# B&R Automation Studio project Panasonic_LinkaPowerCP2_A2021055 (part 42)

#### Main.st - Init, cyclic, exit code
```iecst
PROGRAM _INIT
	(* Insert code here *)
	SKTcpClientTrace_1.Params.IPportClient := 15000;
	SKTcpClientTrace_1.Cmd.LoggerOn:= FALSE;
END_PROGRAM

PROGRAM _CYCLIC

	//Priradenie indexu paletky//
    a:= P2_StoperZaklTesnenia.PAR.CisloPaletky;
	P2_StoperZaklTesnenia.PAR.CisloPaletky_STRING:= USINT_TO_STRING(a);

    //Parametre komunikácie//
    memcpy(ADR(SKTcpClientTrace_1.Params.IPaddrServ),ADR('192.168.128.250'),SIZEOF('192.168.128.250'));

    SKTcpClientTrace_1.Params.IPportServ := 12000;

	SKTcpClientTrace_1.pDevice := ADR('HDD_LOGGER');
	SKTcpClientTrace_1.pFile := ADR('logger_sktcpclienttrace_3.log');
    SKTcpClientTrace_1();

    //Parametre komunikácie//
    //Vstupy pre server//
    SKTcpClientTrace_1.Params.Packet.type := TRCB_P2_ZakladacTesnenia_ST3.INPUTS.TYP_Prikazu;
    SKTcpClientTrace_1.Params.Packet.workplace := TRCB_P2_ZakladacTesnenia_ST3.INPUTS.CisloStanice;
    SKTcpClientTrace_1.Params.Packet.rfid := TRCB_P2_ZakladacTesnenia_ST3.INPUTS.CisloPaletky;
    SKTcpClientTrace_1.Params.Packet.master := TRCB_P2_ZakladacTesnenia_ST3.INPUTS.QRkodPowerCP;
    SKTcpClientTrace_1.Params.Packet.dps1:= TRCB_P2_ZakladacTesnenia_ST3.INPUTS.QRkodFiltra;
    SKTcpClientTrace_1.Params.Packet.dps2:= '';
    SKTcpClientTrace_1.Params.Packet.dps3:= '';
    SKTcpClientTrace_1.Params.Packet.dps4:= '';
    SKTcpClientTrace_1.Params.Packet.dps5:= '';
    SKTcpClientTrace_1.Params.Packet.operator_id := TRCB_P2_ZakladacTesnenia_ST3.INPUTS.ID_Operatora;
    SKTcpClientTrace_1.Params.Packet.data_report:= TRCB_P2_ZakladacTesnenia_ST3.INPUTS.Report;
    SKTcpClientTrace_1.Params.Packet.result := TRCB_P2_ZakladacTesnenia_ST3.INPUTS.StavPaletky;

    //Výstupy zo servera//
    TRCB_P2_ZakladacTesnenia_ST3.OUTPUTS.TYP_Prikazu:= SKTcpClientTrace_1.Internal.Splitter.out[1];
    TRCB_P2_ZakladacTesnenia_ST3.OUTPUTS.CisloStanice:= SKTcpClientTrace_1.Internal.Splitter.out[2];
    TRCB_P2_ZakladacTesnenia_ST3.OUTPUTS.CisloPaletky:= SKTcpClientTrace_1.Internal.Splitter.out[3];
    IF TRCB_P2_ZakladacTesnenia_ST3.INPUTS.TYP_Prikazu = '0' THEN
        TRCB_P2_ZakladacTesnenia_ST3.OUTPUTS.CisloEtikety:= SKTcpClientTrace_1.Internal.Splitter.out[4];
    ELSE
        TRCB_P2_ZakladacTesnenia_ST3.OUTPUTS.QRkodPowerCP:= SKTcpClientTrace_1.Internal.Splitter.out[4];
    END_IF
    TRCB_P2_ZakladacTesnenia_ST3.OUTPUTS.QRkodFiltra:= SKTcpClientTrace_1.Internal.Splitter.out[5];
    TRCB_P2_ZakladacTesnenia_ST3.OUTPUTS.ID_Operatora:= SKTcpClientTrace_1.Internal.Splitter.out[10];
    TRCB_P2_ZakladacTesnenia_ST3.OUTPUTS.DruhCinnostiNaPaletke:= SKTcpClientTrace_1.Internal.Splitter.out[11];
    TRCB_P2_ZakladacTesnenia_ST3.OUTPUTS.PovolenieCinnostiNaPaletke:= SKTcpClientTrace_1.Internal.Splitter.out[12];

    //Volanie funkcie SequenceControl//
    SequenceControl(SC:= SC_KOM_Server);

    CASE SC_KOM_Server.Step OF

        0:
            SC_KOM_Server.StepName:= '0 - Nulovanie';
            SKTcpClientTrace_1.Cmd.Send:= FALSE;
            TRCB_P2_ZakladacTesnenia_ST3.CMD.VyziadajStavPaletky_TYP1:= FALSE;
            TRCB_P2_ZakladacTesnenia_ST3.CMD.PriradQRkodFiltra_TYP3:= FALSE;
            TRCB_P2_ZakladacTesnenia_ST3.CMD.VyziadajCisloEtikety_TYP0:= FALSE;
			TRCB_P2_ZakladacTesnenia_ST3.CMD.OdosliStavPaletky_TYP2:= FALSE;
			TRCB_P2_ZakladacTesnenia_ST3.CMD.VyziadajStavPanatrace_TYP4:= FALSE;
            TRCB_P2_ZakladacTesnenia_ST3.STATUS.KomunikaciaUkoncena:= FALSE;
			TRCB_P2_ZakladacTesnenia_ST3.STATUS.KomunikaciaError:= FALSE;
			TRCB_P2_ZakladacTesnenia_ST3.STATUS.KOM_READY:= FALSE;
            PocetDopytovNaServer:= 0;

            IF SKTcpClientTrace_1.Internal.Step = 0 THEN
                SKTcpClientTrace_1.Enable:= TRUE;
                SC_KOM_Server.ResetStep:= TRUE;
                SC_KOM_Server.Step:= 1;
            ELSIF SKTcpClientTrace_1.Internal.Step = 15 THEN
                SKTcpClientTrace_1.Enable:= TRUE;
                SC_KOM_Server.ResetStep:= TRUE;
                SC_KOM_Server.Step:= 1;
            ELSE
                SKTcpClientTrace_1.Enable:= FALSE;
            END_IF

        1:
            SC_KOM_Server.StepName:= '1 - Rozhodnutie o cinnosti';
            TRCB_P2_ZakladacTesnenia_ST3.STATUS.KOM_READY:= TRUE;
			IF TRCB_P2_ZakladacTesnenia_ST3.CMD.VyziadajStavPaletky_TYP1 THEN
                TRCB_P2_ZakladacTesnenia_ST3.STATUS.KOM_READY:= FALSE;
				SC_KOM_Server.Step:= 10;
            ELSIF TRCB_P2_ZakladacTesnenia_ST3.CMD.PriradQRkodFiltra_TYP3 THEN
                TRCB_P2_ZakladacTesnenia_ST3.STATUS.KOM_READY:= FALSE;
				SC_KOM_Server.Step:= 20;
            ELSIF TRCB_P2_ZakladacTesnenia_ST3.CMD.VyziadajCisloEtikety_TYP0 THEN
                TRCB_P2_ZakladacTesnenia_ST3.STATUS.KOM_READY:= FALSE;
				SC_KOM_Server.Step:= 30;
            ELSIF TRCB_P2_ZakladacTesnenia_ST3.CMD.OdosliStavPaletky_TYP2 THEN
				TRCB_P2_ZakladacTesnenia_ST3.STATUS.KOM_READY:= FALSE;
				SC_KOM_Server.Step:= 40;
			ELSIF TRCB_P2_ZakladacTesnenia_ST3.CMD.VyziadajStavPanatrace_TYP4 THEN
				TRCB_P2_ZakladacTesnenia_ST3.STATUS.KOM_READY:= FALSE;
				SC_KOM_Server.Step:= 50;
            END_IF

        10:
            SC_KOM_Server.StepName:= '10 - Vyziadanie stavu paletky - odoslanie dat na server';
            SC_KOM_Server.IdleTime.PT:= T#3s;
            SC_KOM_Server.AlarmTime.PT:= T#10s;
		    SC_KOM_Server.AlarmTime.IN:= TRUE;

			TRCB_P2_ZakladacTesnenia_ST3.INPUTS.CisloPaletky:= 'Pal';
			brsstrcat(ADR(TRCB_P2_ZakladacTesnenia_ST3.INPUTS.CisloPaletky), ADR(P2_StoperZaklTesnenia.PAR.CisloPaletky_STRING));

            TRCB_P2_ZakladacTesnenia_ST3.INPUTS.TYP_Prikazu:= '1';
            TRCB_P2_ZakladacTesnenia_ST3.INPUTS.CisloStanice:= 'ST3';
            TRCB_P2_ZakladacTesnenia_ST3.INPUTS.QRkodPowerCP:= Paletka[a].PAR.QRkodPowerCP;
            TRCB_P2_ZakladacTesnenia_ST3.INPUTS.QRkodFiltra:= '';
            TRCB_P2_ZakladacTesnenia_ST3.INPUTS.ID_Operatora:= Paletka[a].PAR.ID_Operatora;
            TRCB_P2_ZakladacTesnenia_ST3.INPUTS.Report:= '';
            TRCB_P2_ZakladacTesnenia_ST3.INPUTS.StavPaletky:= 'OK';

			IF SKTcpClientTrace_1.Status.staReadyToSend AND NOT SKTcpClientTrace_1.Cmd.Close THEN
				TRCB_P2_ZakladacTesnenia_ST3.OUTPUTS.TYP_Prikazu:= '';
				SKTcpClientTrace_1.Cmd.Send:= TRUE;
				SC_KOM_Server.ResetStep:= TRUE;
				SC_KOM_Server.Step:= 13;
			END_IF

        13:
			SC_KOM_Server.StepName:= '13 - Vyziadanie stavu paletky - odpoved servera';
            SC_KOM_Server.IdleTime.PT:= T#3s;
            SC_KOM_Server.AlarmTime.PT:= T#7s;
            SC_KOM_Server.AlarmTime.IN:= TRUE;

            IF SKTcpClientTrace_1.Status.staReceived AND
                (TRCB_P2_ZakladacTesnenia_ST3.OUTPUTS.TYP_Prikazu = TRCB_P2_ZakladacTesnenia_ST3.INPUTS.TYP_Prikazu) AND
                (TRCB_P2_ZakladacTesnenia_ST3.OUTPUTS.QRkodPowerCP = TRCB_P2_ZakladacTesnenia_ST3.INPUTS.QRkodPowerCP) THEN
                TRCB_P2_ZakladacTesnenia_ST3.STATUS.KomunikaciaUkoncena:= TRUE;
                SC_KOM_Server.ResetStep:= TRUE;
                SC_KOM_Server.Step:= 15;
            ELSIF SC_KOM_Server.AlarmTime.Q AND NOT SKTcpClientTrace_1.Status.staSending THEN
                PocetDopytovNaServer:= PocetDopytovNaServer + 1;
				SKTcpClientTrace_1.Cmd.Close:= TRUE;
				SKTcpClientTrace_1.Cmd.Send:= FALSE;
				SC_KOM_Server.ResetStep:= TRUE;
                SC_KOM_Server.Step:= 14;
            END_IF

        14:
            SC_KOM_Server.StepName:= '14 - Vyziadanie stavu paletky - cakam na opatovny dopyt na server';
            SC_KOM_Server.IdleTime.PT:= T#1s;
            SC_KOM_Server.AlarmTime.PT:= T#10s;
            SC_KOM_Server.IdleTime.IN:= TRUE;

            IF PocetDopytovNaServer < 3 THEN
                IF SC_KOM_Server.IdleTime.Q THEN
                    SC_KOM_Server.ResetStep:= TRUE;
                    SC_KOM_Server.Step:= 10;
                END_IF
            ELSE
                TRCB_P2_ZakladacTesnenia_ST3.STATUS.KomunikaciaError:= TRUE;
                SC_KOM_Server.ResetStep:= TRUE;
                SC_KOM_Server.Step:= 15;
            END_IF

        15:
            SC_KOM_Server.StepName:= '15 - Vyziadanie stavu paletky - cakam na ukoncenie komunikacie';
            SC_KOM_Server.IdleTime.PT:= T#3s;
            SC_KOM_Server.AlarmTime.PT:= T#10s;

            IF NOT TRCB_P2_ZakladacTesnenia_ST3.CMD.VyziadajStavPaletky_TYP1 THEN
                SC_KOM_Server.ResetStep:= TRUE;
                SC_KOM_Server.Step:= 0;
            END_IF

        20:
            SC_KOM_Server.StepName:= '20 - Priradenie QR kodu - odoslanie dat na server';
            SC_KOM_Server.IdleTime.PT:= T#3s;
            SC_KOM_Server.AlarmTime.PT:= T#20s;
            SC_KOM_Server.AlarmTime.IN:= TRUE;

			TRCB_P2_ZakladacTesnenia_ST3.INPUTS.CisloPaletky:= 'Pal';
			brsstrcat(ADR(TRCB_P2_ZakladacTesnenia_ST3.INPUTS.CisloPaletky), ADR(P2_StoperZaklTesnenia.PAR.CisloPaletky_STRING));

            TRCB_P2_ZakladacTesnenia_ST3.INPUTS.TYP_Prikazu:= '3';
            TRCB_P2_ZakladacTesnenia_ST3.INPUTS.CisloStanice:= 'ST3';
            TRCB_P2_ZakladacTesnenia_ST3.INPUTS.QRkodPowerCP:= Paletka[a].PAR.QRkodPowerCP;
            TRCB_P2_ZakladacTesnenia_ST3.INPUTS.QRkodFiltra:= Paletka[a].PAR.QRkodFiltra_5H;
            TRCB_P2_ZakladacTesnenia_ST3.INPUTS.ID_Operatora:= Paletka[a].PAR.ID_Operatora;
            TRCB_P2_ZakladacTesnenia_ST3.INPUTS.Report:= '';
            TRCB_P2_ZakladacTesnenia_ST3.INPUTS.StavPaletky:= 'OK';

			IF SKTcpClientTrace_1.Status.staReadyToSend AND NOT SKTcpClientTrace_1.Cmd.Close THEN
				TRCB_P2_ZakladacTesnenia_ST3.OUTPUTS.TYP_Prikazu:= '';
				SKTcpClientTrace_1.Cmd.Send:= TRUE;
				SC_KOM_Server.ResetStep:= TRUE;
				SC_KOM_Server.Step:= 23;
			END_IF

        23:
            SC_KOM_Server.StepName:= '23 - Priradenie QR kodu - odpoved servera';
			SC_KOM_Server.IdleTime.PT:= T#3s;
            SC_KOM_Server.AlarmTime.PT:= T#7s;
            SC_KOM_Server.AlarmTime.IN:= TRUE;

            IF SKTcpClientTrace_1.Status.staReceived AND
                (TRCB_P2_ZakladacTesnenia_ST3.OUTPUTS.TYP_Prikazu = TRCB_P2_ZakladacTesnenia_ST3.INPUTS.TYP_Prikazu) AND
                (TRCB_P2_ZakladacTesnenia_ST3.OUTPUTS.QRkodPowerCP = TRCB_P2_ZakladacTesnenia_ST3.INPUTS.QRkodPowerCP) THEN
                TRCB_P2_ZakladacTesnenia_ST3.STATUS.KomunikaciaUkoncena:= TRUE;
                SC_KOM_Server.ResetStep:= TRUE;
                SC_KOM_Server.Step:= 25;
            ELSIF SC_KOM_Server.AlarmTime.Q AND NOT SKTcpClientTrace_1.Status.staSending THEN
                PocetDopytovNaServer:= PocetDopytovNaServer + 1;
				SKTcpClientTrace_1.Cmd.Close:= TRUE;
				SKTcpClientTrace_1.Cmd.Send:= FALSE;
				SC_KOM_Server.ResetStep:= TRUE;
                SC_KOM_Server.Step:= 24;
            END_IF

        24:
            SC_KOM_Server.StepName:= '24 - Priradenie QR kodu - cakam na opatovny dopyt na server';
            SC_KOM_Server.IdleTime.PT:= T#1s;
            SC_KOM_Server.AlarmTime.PT:= T#10s;
            SC_KOM_Server.IdleTime.IN:= TRUE;
            SKTcpClientTrace_1.Cmd.Send:= FALSE;

            IF PocetDopytovNaServer < 3 THEN
                IF SC_KOM_Server.IdleTime.Q THEN
                   	SC_KOM_Server.ResetStep:= TRUE;
                    SC_KOM_Server.Step:= 20;
                END_IF
            ELSE
                TRCB_P2_ZakladacTesnenia_ST3.STATUS.KomunikaciaError:= TRUE;
                SC_KOM_Server.ResetStep:= TRUE;
                SC_KOM_Server.Step:= 25;
            END_IF

        25:
            SC_KOM_Server.StepName:= '25 - Priradenie QR kodu - cakam na ukoncenie komunikacie';
            SC_KOM_Server.IdleTime.PT:= T#3s;
            SC_KOM_Server.AlarmTime.PT:= T#10s;

            IF NOT TRCB_P2_ZakladacTesnenia_ST3.CMD.PriradQRkodFiltra_TYP3 THEN
                SC_KOM_Server.ResetStep:= TRUE;
                SC_KOM_Server.Step:= 0;
            END_IF

        30:
            SC_KOM_Server.StepName:= '30 - Vyziadanie serioveho cisla - odoslanie dat na server';
            SC_KOM_Server.IdleTime.PT:= T#3s;
            SC_KOM_Server.AlarmTime.PT:= T#10s;

            TRCB_P2_ZakladacTesnenia_ST3.INPUTS.TYP_Prikazu:= '0';
            TRCB_P2_ZakladacTesnenia_ST3.INPUTS.CisloStanice:= 'ST3';
            TRCB_P2_ZakladacTesnenia_ST3.INPUTS.CisloPaletky;
            TRCB_P2_ZakladacTesnenia_ST3.INPUTS.QRkodPowerCP:= '';
            TRCB_P2_ZakladacTesnenia_ST3.INPUTS.QRkodFiltra:= '';
            TRCB_P2_ZakladacTesnenia_ST3.INPUTS.ID_Operatora:= 'E2';
            TRCB_P2_ZakladacTesnenia_ST3.INPUTS.Report:= '';
            TRCB_P2_ZakladacTesnenia_ST3.INPUTS.StavPaletky:= 'OK';
            SKTcpClientTrace_1.Cmd.Send:= TRUE;

            IF SKTcpClientTrace_1.Cmd.Send AND NOT SKTcpClientTrace_1.Status.staReceived AND NOT SKTcpClientTrace_1.Status.staError THEN
                SC_KOM_Server.ResetStep:= TRUE;
                SC_KOM_Server.Step:= 33;
            END_IF

        33:
            SC_KOM_Server.StepName:= '33 - Vyziadanie serioveho cisla - odpoved servera';
            SC_KOM_Server.IdleTime.PT:= T#3s;
            SC_KOM_Server.AlarmTime.PT:= T#20s;
            SC_KOM_Server.AlarmTime.IN:= TRUE;

            IF SKTcpClientTrace_1.Status.staReceived AND
                (TRCB_P2_ZakladacTesnenia_ST3.OUTPUTS.TYP_Prikazu = TRCB_P2_ZakladacTesnenia_ST3.INPUTS.TYP_Prikazu) THEN
                TRCB_P2_ZakladacTesnenia_ST3.STATUS.KomunikaciaUkoncena:= TRUE;
                SC_KOM_Server.ResetStep:= TRUE;
                SC_KOM_Server.Step:= 35;
            ELSIF SC_KOM_Server.AlarmTime.Q THEN
                TRCB_P2_ZakladacTesnenia_ST3.STATUS.KomunikaciaError:= TRUE;
                SC_KOM_Server.ResetStep:= TRUE;
                SC_KOM_Server.Step:= 35;
            END_IF

        35:
            SC_KOM_Server.StepName:= '35 - Vyziadanie serioveho cisla - cakam na ukoncenie komunikacie';
            SC_KOM_Server.IdleTime.PT:= T#3s;
            SC_KOM_Server.AlarmTime.PT:= T#10s;

            IF NOT TRCB_P2_ZakladacTesnenia_ST3.CMD.VyziadajCisloEtikety_TYP0 THEN
                SC_KOM_Server.ResetStep:= TRUE;
                SC_KOM_Server.Step:= 0;
            END_IF

        40:
            SC_KOM_Server.StepName:= '40 - Odoslanie stavu paletky - odoslanie dat na server';
            SC_KOM_Server.IdleTime.PT:= T#3s;
            SC_KOM_Server.AlarmTime.PT:= T#20s;
            SC_KOM_Server.AlarmTime.IN:= TRUE;

            //Vytvorenie spravy pre report//

            IF NOT SC_KOM_Server.Switch1 THEN
				brsmemset(ADR(Report),0,SIZEOF(Report));
				brsmemset(ADR(TRCB_P2_ZakladacTesnenia_ST3.INPUTS.Report), 0, SIZEOF(TRCB_P2_ZakladacTesnenia_ST3.INPUTS.Report));

				//Kamera 17 - kontrola paletky//
                Report[0].PoradoveCislo:= '1';
                Report[0].Popis:= 'KAM_17_KontrolaPaletky';
                Report[0].FormatHodnoty:= '2';
                Report[0].Tolerancia_MIN_Hodnota:= '';
                Report[0].Tolerancia_MAX_Hodnota:= '';
                Report[0].Nominal:= 'OK';
                Report[0].Tolerancia_MIN_Jednotky:= '';
                Report[0].Tolerancia_MAX_Jednotky:= '';
                IF Reports.Kamery.P2_CAM17_KontrolaPaletky = 'PASS' THEN
                    Report[0].NameranaHodnota:= 'OK';
                ELSE
                    Report[0].NameranaHodnota:= 'NG';
                END_IF
                Report[0].NameranaHodnota_Jednotky:= '';
                Report[0].VyslednyResult:= Reports.Kamery.P2_CAM17_KontrolaPaletky;
                SKTcpClientNewCsvEntry(Report[0].PoradoveCislo,Report[0].Popis,Report[0].FormatHodnoty,Report[0].Tolerancia_MIN_Hodnota,Report[0].Tolerancia_MAX_Hodnota,Report[0].Nominal,Report[0].Tolerancia_MIN_Jednotky,Report[0].Tolerancia_MAX_Jednotky,Report[0].NameranaHodnota,Report[0].NameranaHodnota_Jednotky,Report[0].VyslednyResult, ADR(TRCB_P2_ZakladacTesnenia_ST3.INPUTS.Report));

                //Kamera 1 - kontrola tesnenia//
                Report[1].PoradoveCislo:= '2';
                Report[1].Popis:= 'KAM_1_KontrolaTesnenia';
                Report[1].FormatHodnoty:= '2';
                Report[1].Tolerancia_MIN_Hodnota:= '';
                Report[1].Tolerancia_MAX_Hodnota:= '';
                Report[1].Nominal:= 'OK';
                Report[1].Tolerancia_MIN_Jednotky:= '';
                Report[1].Tolerancia_MAX_Jednotky:= '';
                IF Reports.Kamery.P2_CAM1_KontrolaTesnenia = 'PASS' THEN
                    Report[1].NameranaHodnota:= 'OK';
                ELSE
                    Report[1].NameranaHodnota:= 'NG';
                END_IF
                Report[1].NameranaHodnota_Jednotky:= '';
                Report[1].VyslednyResult:= Reports.Kamery.P2_CAM1_KontrolaTesnenia;
                SKTcpClientNewCsvEntry(Report[1].PoradoveCislo,Report[1].Popis,Report[1].FormatHodnoty,Report[1].Tolerancia_MIN_Hodnota,Report[1].Tolerancia_MAX_Hodnota,Report[1].Nominal,Report[1].Tolerancia_MIN_Jednotky,Report[1].Tolerancia_MAX_Jednotky,Report[1].NameranaHodnota,Report[1].NameranaHodnota_Jednotky,Report[1].VyslednyResult, ADR(TRCB_P2_ZakladacTesnenia_ST3.INPUTS.Report));
                SC_KOM_Server.Switch1:= TRUE;
            END_IF

			TRCB_P2_ZakladacTesnenia_ST3.INPUTS.CisloPaletky:= 'Pal';
			brsstrcat(ADR(TRCB_P2_ZakladacTesnenia_ST3.INPUTS.CisloPaletky), ADR(P2_StoperZaklTesnenia.PAR.CisloPaletky_STRING));

            TRCB_P2_ZakladacTesnenia_ST3.INPUTS.TYP_Prikazu:= '2';
            TRCB_P2_ZakladacTesnenia_ST3.INPUTS.CisloStanice:= 'ST3';
            TRCB_P2_ZakladacTesnenia_ST3.INPUTS.QRkodPowerCP:= Paletka[a].PAR.QRkodPowerCP;
            TRCB_P2_ZakladacTesnenia_ST3.INPUTS.QRkodFiltra:= '';
            TRCB_P2_ZakladacTesnenia_ST3.INPUTS.ID_Operatora:= Paletka[a].PAR.ID_Operatora;
            TRCB_P2_ZakladacTesnenia_ST3.INPUTS.StavPaletky:= Paletka[a].PAR.StavPowerCP;

			IF SKTcpClientTrace_1.Status.staReadyToSend AND NOT SKTcpClientTrace_1.Cmd.Close THEN
				TRCB_P2_ZakladacTesnenia_ST3.OUTPUTS.TYP_Prikazu:= '';
				SKTcpClientTrace_1.Cmd.Send:= TRUE;
				SC_KOM_Server.ResetStep:= TRUE;
				SC_KOM_Server.Step:= 43;
			END_IF

        43:
            SC_KOM_Server.StepName:= '43 - Odoslanie stavu paletky - odpoved servera';
			SC_KOM_Server.IdleTime.PT:= T#3s;
            SC_KOM_Server.AlarmTime.PT:= T#7s;
            SC_KOM_Server.AlarmTime.IN:= TRUE;

            IF SKTcpClientTrace_1.Status.staReceived AND
                (TRCB_P2_ZakladacTesnenia_ST3.OUTPUTS.TYP_Prikazu = TRCB_P2_ZakladacTesnenia_ST3.INPUTS.TYP_Prikazu) AND
                (TRCB_P2_ZakladacTesnenia_ST3.OUTPUTS.QRkodPowerCP = TRCB_P2_ZakladacTesnenia_ST3.INPUTS.QRkodPowerCP) THEN
                TRCB_P2_ZakladacTesnenia_ST3.STATUS.KomunikaciaUkoncena:= TRUE;
                SC_KOM_Server.ResetStep:= TRUE;
                SC_KOM_Server.Step:= 45;
            ELSIF SC_KOM_Server.AlarmTime.Q AND NOT SKTcpClientTrace_1.Status.staSending THEN
                PocetDopytovNaServer:= PocetDopytovNaServer + 1;
				SKTcpClientTrace_1.Cmd.Close:= TRUE;
				SKTcpClientTrace_1.Cmd.Send:= FALSE;
				SC_KOM_Server.ResetStep:= TRUE;
                SC_KOM_Server.Step:= 44;
            END_IF

        44:
            SC_KOM_Server.StepName:= '44 - Odoslanie stavu paletky - cakam na opatovny dopyt na server';
            SC_KOM_Server.IdleTime.PT:= T#1s;
            SC_KOM_Server.AlarmTime.PT:= T#10s;
            SC_KOM_Server.IdleTime.IN:= TRUE;
            SKTcpClientTrace_1.Cmd.Send:= FALSE;

            IF PocetDopytovNaServer < 3 THEN
                IF SC_KOM_Server.IdleTime.Q THEN
                    SC_KOM_Server.ResetStep:= TRUE;
                    SC_KOM_Server.Step:= 40;
                END_IF
            ELSE
                TRCB_P2_ZakladacTesnenia_ST3.STATUS.KomunikaciaError:= TRUE;
                SC_KOM_Server.ResetStep:= TRUE;
                SC_KOM_Server.Step:= 45;
            END_IF

        45:
            SC_KOM_Server.StepName:= '45 - Odoslanie stavu paletky - cakam na ukoncenie komunikacie';
            SC_KOM_Server.IdleTime.PT:= T#3s;
            SC_KOM_Server.AlarmTime.PT:= T#10s;

            IF NOT TRCB_P2_ZakladacTesnenia_ST3.CMD.OdosliStavPaletky_TYP2 THEN
                SC_KOM_Server.ResetStep:= TRUE;
                SC_KOM_Server.Step:= 0;
            END_IF

		50:
			SC_KOM_Server.StepName:= '50 - Vyziadanie stavu Panatrace - odoslanie dat na server';
			SC_KOM_Server.IdleTime.PT:= T#3s;
			SC_KOM_Server.AlarmTime.PT:= T#10s;
			SC_KOM_Server.AlarmTime.IN:= TRUE;

			TRCB_P2_ZakladacTesnenia_ST3.INPUTS.TYP_Prikazu:= '4';
			TRCB_P2_ZakladacTesnenia_ST3.INPUTS.CisloStanice:= 'ST3';
			TRCB_P2_ZakladacTesnenia_ST3.INPUTS.CisloPaletky:= '';
			TRCB_P2_ZakladacTesnenia_ST3.INPUTS.QRkodPowerCP:= '';
			TRCB_P2_ZakladacTesnenia_ST3.INPUTS.QRkodFiltra:= '';
			TRCB_P2_ZakladacTesnenia_ST3.INPUTS.ID_Operatora:= '';
			TRCB_P2_ZakladacTesnenia_ST3.INPUTS.Report:= '';
			TRCB_P2_ZakladacTesnenia_ST3.INPUTS.StavPaletky:= '';

			IF SKTcpClientTrace_1.Status.staReadyToSend AND NOT SKTcpClientTrace_1.Cmd.Close THEN
				TRCB_P2_ZakladacTesnenia_ST3.OUTPUTS.TYP_Prikazu:= '';
				SKTcpClientTrace_1.Cmd.Send:= TRUE;
				SC_KOM_Server.ResetStep:= TRUE;
				SC_KOM_Server.Step:= 53;
			END_IF

		53:
			SC_KOM_Server.StepName:= '53 - Vyziadanie stavu paletky - odpoved servera';
			SC_KOM_Server.IdleTime.PT:= T#30s;
			SC_KOM_Server.AlarmTime.PT:= T#7s;
			SC_KOM_Server.AlarmTime.IN:= TRUE;

			IF SKTcpClientTrace_1.Status.staReceived AND TRCB_P2_ZakladacTesnenia_ST3.OUTPUTS.TYP_Prikazu = TRCB_P2_ZakladacTesnenia_ST3.INPUTS.TYP_Prikazu THEN
				TRCB_P2_ZakladacTesnenia_ST3.STATUS.KomunikaciaUkoncena:= TRUE;
				SC_KOM_Server.ResetStep:= TRUE;
				SC_KOM_Server.Step:= 55;
			ELSIF SC_KOM_Server.AlarmTime.Q AND NOT SKTcpClientTrace_1.Status.staSending THEN
				PocetDopytovNaServer:= PocetDopytovNaServer + 1;
				SKTcpClientTrace_1.Cmd.Close:= TRUE;
				SKTcpClientTrace_1.Cmd.Send:= FALSE;
				SC_KOM_Server.ResetStep:= TRUE;
				SC_KOM_Server.Step:= 54;
			END_IF

		54:
			SC_KOM_Server.StepName:= '54 - Vyziadanie stavu paletky - cakam na opatovny dopyt na server';
			SC_KOM_Server.IdleTime.PT:= T#1s;
			SC_KOM_Server.AlarmTime.PT:= T#10s;
			SC_KOM_Server.IdleTime.IN:= TRUE;

			IF PocetDopytovNaServer < 3 THEN
				IF SC_KOM_Server.IdleTime.Q THEN
					SC_KOM_Server.ResetStep:= TRUE;
					SC_KOM_Server.Step:= 50;
				END_IF
			ELSE
				TRCB_P2_ZakladacTesnenia_ST3.STATUS.KomunikaciaError:= TRUE;
				SC_KOM_Server.ResetStep:= TRUE;
				SC_KOM_Server.Step:= 55;
			END_IF

		55:
			SC_KOM_Server.StepName:= '55 - Vyziadanie stavu paletky - cakam na ukoncenie komunikacie';
			SC_KOM_Server.IdleTime.PT:= T#3s;
			SC_KOM_Server.AlarmTime.PT:= T#10s;

			IF NOT TRCB_P2_ZakladacTesnenia_ST3.CMD.VyziadajStavPanatrace_TYP4 THEN
				SC_KOM_Server.ResetStep:= TRUE;
				SC_KOM_Server.Step:= 0;
			END_IF

    END_CASE

END_PROGRAM

PROGRAM _EXIT
	(* Insert code here *)

END_PROGRAM
```

#### Types.typ - Local data types
```iecst
TYPE
	Report_typ : 	STRUCT
		PoradoveCislo : STRING[2]; (*IDstep - Poradové čislo reportu*)
		Popis : STRING[100]; (*Description - Popis*)
		FormatHodnoty : STRING[2]; (*TypValue - Format zaslané hodnoty  1- Číslo, 2 - Znak*)
		Tolerancia_MIN_Hodnota : STRING[10]; (*MinTol - Minimálna tolerancia meranej veličiny*)
		Tolerancia_MAX_Hodnota : STRING[10]; (*MaxTol - Maximálna tolerancia meranej veličiny*)
		Nominal : STRING[10]; (*Nom - Ak jezvolený formát string tak tu zadáme OK inak je prazdna*)
		Tolerancia_MIN_Jednotky : STRING[10]; (*MinEle - Jednotky minimálnej tolerancie veličiny*)
		Tolerancia_MAX_Jednotky : STRING[10]; (*MaxEle - Jednotky maximálnej tolerancie veličiny*)
		NameranaHodnota : STRING[10]; (*Value - Namerana hodnota veličiny, ak su kamery tak bude hodnota OK alebo NG*)
		NameranaHodnota_Jednotky : STRING[10]; (*ValEle - Jednotky nameranej veličiny*)
		VyslednyResult : STRING[5]; (*Result - Výsledný result  PASS, FAIL, SKIP*)
	END_STRUCT;
END_TYPE
```

#### Variables.var - Local variables
```iecst
VAR
	SC_KOM_Server : SequenceControlTyp;
	SKTcpClientTrace_1 : SKTcpClientTrace;
	a : USINT;
	Report : ARRAY[0..50] OF Report_typ;
	PocetDopytovNaServer : USINT;
END_VAR
```

### Program Logical/TracebilitySystem/P2_Maticovacka_ST4 (IEC)

#### Main.st - Init, cyclic, exit code
```iecst
PROGRAM _INIT
	(* Insert code here *)
	SKTcpClientTrace_1.Params.IPportClient := 16000;
	SKTcpClientTrace_1.Cmd.LoggerOn:= FALSE;
END_PROGRAM

PROGRAM _CYCLIC

	//Priradenie indexu paletky//
	a:= P2_StoperMaticovacky.PAR.CisloPaletky;
	P2_StoperMaticovacky.PAR.CisloPaletky_STRING:= USINT_TO_STRING(a);

	//Parametre komunikácie//
	memcpy(ADR(SKTcpClientTrace_1.Params.IPaddrServ),ADR('192.168.128.250'),SIZEOF('192.168.128.250'));

    SKTcpClientTrace_1.Params.IPportServ := 12000;

	SKTcpClientTrace_1.pDevice := ADR('HDD_LOGGER');
	SKTcpClientTrace_1.pFile := ADR('logger_sktcpclienttrace_4.log');
	SKTcpClientTrace_1();

	//Parametre komunikácie//
	//Vstupy pre server//
	SKTcpClientTrace_1.Params.Packet.type := TRCB_P2_Maticovacka_ST4.INPUTS.TYP_Prikazu;
	SKTcpClientTrace_1.Params.Packet.workplace := TRCB_P2_Maticovacka_ST4.INPUTS.CisloStanice;
	SKTcpClientTrace_1.Params.Packet.rfid := TRCB_P2_Maticovacka_ST4.INPUTS.CisloPaletky;
	SKTcpClientTrace_1.Params.Packet.master := TRCB_P2_Maticovacka_ST4.INPUTS.QRkodPowerCP;
	SKTcpClientTrace_1.Params.Packet.dps1:= TRCB_P2_Maticovacka_ST4.INPUTS.QRkodFiltra;
	SKTcpClientTrace_1.Params.Packet.dps2:= '';
	SKTcpClientTrace_1.Params.Packet.dps3:= '';
	SKTcpClientTrace_1.Params.Packet.dps4:= '';
	SKTcpClientTrace_1.Params.Packet.dps5:= '';
	SKTcpClientTrace_1.Params.Packet.operator_id := TRCB_P2_Maticovacka_ST4.INPUTS.ID_Operatora;
	SKTcpClientTrace_1.Params.Packet.data_report:= TRCB_P2_Maticovacka_ST4.INPUTS.Report;
	SKTcpClientTrace_1.Params.Packet.result := TRCB_P2_Maticovacka_ST4.INPUTS.StavPaletky;

	//Výstupy zo servera//
	TRCB_P2_Maticovacka_ST4.OUTPUTS.TYP_Prikazu:= SKTcpClientTrace_1.Internal.Splitter.out[1];
	TRCB_P2_Maticovacka_ST4.OUTPUTS.CisloStanice:= SKTcpClientTrace_1.Internal.Splitter.out[2];
	TRCB_P2_Maticovacka_ST4.OUTPUTS.CisloPaletky:= SKTcpClientTrace_1.Internal.Splitter.out[3];
	IF TRCB_P2_Maticovacka_ST4.INPUTS.TYP_Prikazu = '0' THEN
		TRCB_P2_Maticovacka_ST4.OUTPUTS.CisloEtikety:= SKTcpClientTrace_1.Internal.Splitter.out[4];
	ELSE
		TRCB_P2_Maticovacka_ST4.OUTPUTS.QRkodPowerCP:= SKTcpClientTrace_1.Internal.Splitter.out[4];
	END_IF
	TRCB_P2_Maticovacka_ST4.OUTPUTS.QRkodFiltra:= SKTcpClientTrace_1.Internal.Splitter.out[5];
	TRCB_P2_Maticovacka_ST4.OUTPUTS.ID_Operatora:= SKTcpClientTrace_1.Internal.Splitter.out[10];
	TRCB_P2_Maticovacka_ST4.OUTPUTS.DruhCinnostiNaPaletke:= SKTcpClientTrace_1.Internal.Splitter.out[11];
	TRCB_P2_Maticovacka_ST4.OUTPUTS.PovolenieCinnostiNaPaletke:= SKTcpClientTrace_1.Internal.Splitter.out[12];

	//Volanie funkcie SequenceControl//
	SequenceControl(SC:= SC_KOM_Server);

    CASE SC_KOM_Server.Step OF

        0:
			SC_KOM_Server.StepName:= '0 - Nulovanie';
			SKTcpClientTrace_1.Cmd.Send:= FALSE;
			TRCB_P2_Maticovacka_ST4.CMD.VyziadajStavPaletky_TYP1:= FALSE;
			TRCB_P2_Maticovacka_ST4.CMD.PriradQRkodFiltra_TYP3:= FALSE;
			TRCB_P2_Maticovacka_ST4.CMD.VyziadajCisloEtikety_TYP0:= FALSE;
			TRCB_P2_Maticovacka_ST4.CMD.OdosliStavPaletky_TYP2:= FALSE;
			TRCB_P2_Maticovacka_ST4.CMD.VyziadajStavPanatrace_TYP4:= FALSE;
            TRCB_P2_Maticovacka_ST4.STATUS.KomunikaciaUkoncena:= FALSE;
			TRCB_P2_Maticovacka_ST4.STATUS.KomunikaciaError:= FALSE;
			TRCB_P2_Maticovacka_ST4.STATUS.KOM_READY:= FALSE;
            PocetDopytovNaServer:= 0;

			IF SKTcpClientTrace_1.Internal.Step = 0 THEN
				SKTcpClientTrace_1.Enable:= TRUE;
				SC_KOM_Server.ResetStep:= TRUE;
				SC_KOM_Server.Step:= 1;
			ELSIF SKTcpClientTrace_1.Internal.Step = 15 THEN
				SKTcpClientTrace_1.Enable:= TRUE;
				SC_KOM_Server.ResetStep:= TRUE;
				SC_KOM_Server.Step:= 1;
			ELSE
				SKTcpClientTrace_1.Enable:= FALSE;
			END_IF

		1:
			SC_KOM_Server.StepName:= '1 - Rozhodnutie o cinnosti';
			TRCB_P2_Maticovacka_ST4.STATUS.KOM_READY:= TRUE;
			IF TRCB_P2_Maticovacka_ST4.CMD.VyziadajStavPaletky_TYP1 THEN
				TRCB_P2_Maticovacka_ST4.STATUS.KOM_READY:= FALSE;
				SC_KOM_Server.Step:= 10;
			ELSIF TRCB_P2_Maticovacka_ST4.CMD.PriradQRkodFiltra_TYP3 THEN
				TRCB_P2_Maticovacka_ST4.STATUS.KOM_READY:= FALSE;
				SC_KOM_Server.Step:= 20;
			ELSIF TRCB_P2_Maticovacka_ST4.CMD.VyziadajCisloEtikety_TYP0 THEN
				TRCB_P2_Maticovacka_ST4.STATUS.KOM_READY:= FALSE;
				SC_KOM_Server.Step:= 30;
			ELSIF TRCB_P2_Maticovacka_ST4.CMD.OdosliStavPaletky_TYP2 THEN
				TRCB_P2_Maticovacka_ST4.STATUS.KOM_READY:= FALSE;
				SC_KOM_Server.Step:= 40;
			ELSIF TRCB_P2_Maticovacka_ST4.CMD.VyziadajStavPanatrace_TYP4 THEN
				TRCB_P2_Maticovacka_ST4.STATUS.KOM_READY:= FALSE;
				SC_KOM_Server.Step:= 50;
			END_IF

		10:
			SC_KOM_Server.StepName:= '10 - Vyziadanie stavu paletky - odoslanie dat na server';
			SC_KOM_Server.IdleTime.PT:= T#3s;
            SC_KOM_Server.AlarmTime.PT:= T#5s;
            SC_KOM_Server.AlarmTime.IN:= TRUE;

			TRCB_P2_Maticovacka_ST4.INPUTS.CisloPaletky:= 'Pal';
			brsstrcat(ADR(TRCB_P2_Maticovacka_ST4.INPUTS.CisloPaletky), ADR(P2_StoperMaticovacky.PAR.CisloPaletky_STRING));

			TRCB_P2_Maticovacka_ST4.INPUTS.TYP_Prikazu:= '1';
			TRCB_P2_Maticovacka_ST4.INPUTS.CisloStanice:= 'ST4';
			TRCB_P2_Maticovacka_ST4.INPUTS.QRkodPowerCP:= Paletka[a].PAR.QRkodPowerCP;
			TRCB_P2_Maticovacka_ST4.INPUTS.QRkodFiltra:= '';
			TRCB_P2_Maticovacka_ST4.INPUTS.ID_Operatora:= Paletka[a].PAR.ID_Operatora;
			TRCB_P2_Maticovacka_ST4.INPUTS.Report:= '';
			TRCB_P2_Maticovacka_ST4.INPUTS.StavPaletky:= 'OK';

			IF SKTcpClientTrace_1.Status.staReadyToSend AND NOT SKTcpClientTrace_1.Cmd.Close THEN
				TRCB_P2_Maticovacka_ST4.OUTPUTS.TYP_Prikazu:= '';
				SKTcpClientTrace_1.Cmd.Send:= TRUE;
				SC_KOM_Server.ResetStep:= TRUE;
				SC_KOM_Server.Step:= 13;
			END_IF

		13:
			SC_KOM_Server.StepName:= '13 - Vyziadanie stavu paletky - odpoved servera';
			SC_KOM_Server.IdleTime.PT:= T#3s;
            SC_KOM_Server.AlarmTime.PT:= T#7s;
            SC_KOM_Server.AlarmTime.IN:= TRUE;

			IF SKTcpClientTrace_1.Status.staReceived AND
				(TRCB_P2_Maticovacka_ST4.OUTPUTS.TYP_Prikazu = TRCB_P2_Maticovacka_ST4.INPUTS.TYP_Prikazu) AND
				(TRCB_P2_Maticovacka_ST4.OUTPUTS.QRkodPowerCP = TRCB_P2_Maticovacka_ST4.INPUTS.QRkodPowerCP) THEN
				TRCB_P2_Maticovacka_ST4.STATUS.KomunikaciaUkoncena:= TRUE;
				SC_KOM_Server.ResetStep:= TRUE;
				SC_KOM_Server.Step:= 15;
            ELSIF SC_KOM_Server.AlarmTime.Q AND NOT SKTcpClientTrace_1.Status.staSending THEN
                PocetDopytovNaServer:= PocetDopytovNaServer + 1;
				SKTcpClientTrace_1.Cmd.Close:= TRUE;
				SKTcpClientTrace_1.Cmd.Send:= FALSE;
				SC_KOM_Server.ResetStep:= TRUE;
                SC_KOM_Server.Step:= 14;
            END_IF

        14:
            SC_KOM_Server.StepName:= '14 - Vyziadanie stavu paletky - cakam na opatovny dopyt na server';
            SC_KOM_Server.IdleTime.PT:= T#1s;
            SC_KOM_Server.AlarmTime.PT:= T#10s;
            SC_KOM_Server.IdleTime.IN:= TRUE;

            IF PocetDopytovNaServer < 3 THEN
                IF SC_KOM_Server.IdleTime.Q THEN
                    SC_KOM_Server.ResetStep:= TRUE;
                    SC_KOM_Server.Step:= 10;
                END_IF
            ELSE
                TRCB_P2_Maticovacka_ST4.STATUS.KomunikaciaError:= TRUE;
                SC_KOM_Server.ResetStep:= TRUE;
                SC_KOM_Server.Step:= 15;
            END_IF

		15:
			SC_KOM_Server.StepName:= '15 - Vyziadanie stavu paletky - cakam na ukoncenie komunikacie';
			SC_KOM_Server.IdleTime.PT:= T#3s;
			SC_KOM_Server.AlarmTime.PT:= T#10s;

			IF NOT TRCB_P2_Maticovacka_ST4.CMD.VyziadajStavPaletky_TYP1 THEN
                SC_KOM_Server.ResetStep:= TRUE;
				SC_KOM_Server.Step:= 0;
			END_IF

		20:
			SC_KOM_Server.StepName:= '20 - Priradenie QR kodu - odoslanie dat na server';
			SC_KOM_Server.IdleTime.PT:= T#3s;
			SC_KOM_Server.AlarmTime.PT:= T#10s;

			TRCB_P2_Maticovacka_ST4.INPUTS.TYP_Prikazu:= '3';
			TRCB_P2_Maticovacka_ST4.INPUTS.CisloStanice:= 'ST4';
			TRCB_P2_Maticovacka_ST4.INPUTS.CisloPaletky;
			TRCB_P2_Maticovacka_ST4.INPUTS.QRkodPowerCP:= Paletka[a].PAR.QRkodPowerCP;
			TRCB_P2_Maticovacka_ST4.INPUTS.QRkodFiltra:= '';
			TRCB_P2_Maticovacka_ST4.INPUTS.ID_Operatora:= Paletka[a].PAR.ID_Operatora;
			TRCB_P2_Maticovacka_ST4.INPUTS.Report:= '';
			TRCB_P2_Maticovacka_ST4.INPUTS.StavPaletky:= 'OK';
			SKTcpClientTrace_1.Cmd.Send:= TRUE;

			IF SKTcpClientTrace_1.Cmd.Send AND NOT SKTcpClientTrace_1.Status.staReceived AND NOT SKTcpClientTrace_1.Status.staError THEN
				SC_KOM_Server.ResetStep:= TRUE;
				SC_KOM_Server.Step:= 23;
			END_IF

		23:
			SC_KOM_Server.StepName:= '23 - Priradenie QR kodu - odpoved servera';
			SC_KOM_Server.IdleTime.PT:= T#3s;
            SC_KOM_Server.AlarmTime.PT:= T#20s;
            SC_KOM_Server.AlarmTime.IN:= TRUE;

			IF SKTcpClientTrace_1.Status.staReceived AND
				(TRCB_P2_Maticovacka_ST4.OUTPUTS.TYP_Prikazu = TRCB_P2_Maticovacka_ST4.INPUTS.TYP_Prikazu) AND
				(TRCB_P2_Maticovacka_ST4.OUTPUTS.QRkodPowerCP = TRCB_P2_Maticovacka_ST4.INPUTS.QRkodPowerCP) THEN
				TRCB_P2_Maticovacka_ST4.STATUS.KomunikaciaUkoncena:= TRUE;
				SC_KOM_Server.ResetStep:= TRUE;
                SC_KOM_Server.Step:= 25;
            ELSIF SC_KOM_Server.AlarmTime.Q THEN
                TRCB_P2_Maticovacka_ST4.STATUS.KomunikaciaError:= TRUE;
                SC_KOM_Server.ResetStep:= TRUE;
                SC_KOM_Server.Step:= 25;
			END_IF

		25:
			SC_KOM_Server.StepName:= '25 - Priradenie QR kodu - cakam na ukoncenie komunikacie';
			SC_KOM_Server.IdleTime.PT:= T#3s;
			SC_KOM_Server.AlarmTime.PT:= T#10s;

			IF NOT TRCB_P2_Maticovacka_ST4.CMD.PriradQRkodFiltra_TYP3 THEN
                SC_KOM_Server.ResetStep:= TRUE;
				SC_KOM_Server.Step:= 0;
			END_IF

		30:
			SC_KOM_Server.StepName:= '30 - Vyziadanie serioveho cisla - odoslanie dat na server';
			SC_KOM_Server.IdleTime.PT:= T#3s;
			SC_KOM_Server.AlarmTime.PT:= T#10s;

			TRCB_P2_Maticovacka_ST4.INPUTS.TYP_Prikazu:= '0';
			TRCB_P2_Maticovacka_ST4.INPUTS.CisloStanice:= 'ST4';
			TRCB_P2_Maticovacka_ST4.INPUTS.CisloPaletky;
			TRCB_P2_Maticovacka_ST4.INPUTS.QRkodPowerCP:= '';
			TRCB_P2_Maticovacka_ST4.INPUTS.QRkodFiltra:= '';
			TRCB_P2_Maticovacka_ST4.INPUTS.ID_Operatora:= 'E2';
			TRCB_P2_Maticovacka_ST4.INPUTS.Report:= '';
			TRCB_P2_Maticovacka_ST4.INPUTS.StavPaletky:= 'OK';
			SKTcpClientTrace_1.Cmd.Send:= TRUE;

			IF SKTcpClientTrace_1.Cmd.Send AND NOT SKTcpClientTrace_1.Status.staReceived AND NOT SKTcpClientTrace_1.Status.staError THEN
				SC_KOM_Server.ResetStep:= TRUE;
				SC_KOM_Server.Step:= 33;
			END_IF

		33:
			SC_KOM_Server.StepName:= '33 - Vyziadanie serioveho cisla - odpoved servera';
			SC_KOM_Server.IdleTime.PT:= T#3s;
            SC_KOM_Server.AlarmTime.PT:= T#20s;
            SC_KOM_Server.AlarmTime.IN:= TRUE;

			IF SKTcpClientTrace_1.Status.staReceived AND
				(TRCB_P2_Maticovacka_ST4.OUTPUTS.TYP_Prikazu = TRCB_P2_Maticovacka_ST4.INPUTS.TYP_Prikazu) THEN
				TRCB_P2_Maticovacka_ST4.STATUS.KomunikaciaUkoncena:= TRUE;
				SC_KOM_Server.ResetStep:= TRUE;
                SC_KOM_Server.Step:= 35;
           ELSIF SC_KOM_Server.AlarmTime.Q THEN
                TRCB_P2_Maticovacka_ST4.STATUS.KomunikaciaError:= TRUE;
                SC_KOM_Server.ResetStep:= TRUE;
                SC_KOM_Server.Step:= 35;
			END_IF

		35:
			SC_KOM_Server.StepName:= '35 - Vyziadanie serioveho cisla - cakam na ukoncenie komunikacie';
			SC_KOM_Server.IdleTime.PT:= T#3s;
			SC_KOM_Server.AlarmTime.PT:= T#10s;

			IF NOT TRCB_P2_Maticovacka_ST4.CMD.VyziadajCisloEtikety_TYP0 THEN
                SC_KOM_Server.ResetStep:= TRUE;
				SC_KOM_Server.Step:= 0;
			END_IF

		40:
			SC_KOM_Server.StepName:= '40 - Odoslanie stavu paletky - odoslanie dat na server';
			SC_KOM_Server.IdleTime.PT:= T#3s;
            SC_KOM_Server.AlarmTime.PT:= T#20s;
            SC_KOM_Server.AlarmTime.IN:= TRUE;

            //Vytvorenie spravy pre report//
            IF NOT SC_KOM_Server.Switch1 THEN
                brsmemset(ADR(Report),0,SIZEOF(Report));
				brsmemset(ADR(TRCB_P2_Maticovacka_ST4.INPUTS.Report), 0, SIZEOF(TRCB_P2_Maticovacka_ST4.INPUTS.Report));

				//Matica M4 //
                Report[0].PoradoveCislo:= '1';
                Report[0].Popis:= 'MaticaM4_Moment';
                Report[0].FormatHodnoty:= '1';
                Report[0].Tolerancia_MIN_Hodnota:= Reports.Skrutkovacky.Moment_ToleranciaMIN.P2_MaticaM4;
                Report[0].Tolerancia_MAX_Hodnota:= Reports.Skrutkovacky.Moment_ToleranciaMAX.P2_MaticaM4;
                Report[0].Nominal:= '';
                Report[0].Tolerancia_MIN_Jednotky:= 'Nm';
                Report[0].Tolerancia_MAX_Jednotky:= 'Nm';
                Report[0].NameranaHodnota:= Reports.Skrutkovacky.Moment_NameranaHodnota.P2_MaticaM4;
                Report[0].NameranaHodnota_Jednotky:= 'Nm';
                Report[0].VyslednyResult:= Reports.Skrutkovacky.VyslednyReport.P2_MaticaM4;
                SKTcpClientNewCsvEntry(Report[0].PoradoveCislo,Report[0].Popis,Report[0].FormatHodnoty,Report[0].Tolerancia_MIN_Hodnota,Report[0].Tolerancia_MAX_Hodnota,Report[0].Nominal,Report[0].Tolerancia_MIN_Jednotky,Report[0].Tolerancia_MAX_Jednotky,Report[0].NameranaHodnota,Report[0].NameranaHodnota_Jednotky,Report[0].VyslednyResult, ADR(TRCB_P2_Maticovacka_ST4.INPUTS.Report));

                Report[1].PoradoveCislo:= '2';
                Report[1].Popis:= 'MaticaM4_Uhol';
                Report[1].FormatHodnoty:= '1';
                Report[1].Tolerancia_MIN_Hodnota:= Reports.Skrutkovacky.Uhol_ToleranciaMIN.P2_MaticaM4;
                Report[1].Tolerancia_MAX_Hodnota:= Reports.Skrutkovacky.Uhol_ToleranciaMAX.P2_MaticaM4;
                Report[1].Nominal:= '';
                Report[1].Tolerancia_MIN_Jednotky:= 'st';
                Report[1].Tolerancia_MAX_Jednotky:= 'st';
                Report[1].NameranaHodnota:= Reports.Skrutkovacky.Uhol_NameranaHodnota.P2_MaticaM4;
                Report[1].NameranaHodnota_Jednotky:= 'st';
                Report[1].VyslednyResult:= Reports.Skrutkovacky.VyslednyReport.P2_MaticaM4;
                SKTcpClientNewCsvEntry(Report[1].PoradoveCislo,Report[1].Popis,Report[1].FormatHodnoty,Report[1].Tolerancia_MIN_Hodnota,Report[1].Tolerancia_MAX_Hodnota,Report[1].Nominal,Report[1].Tolerancia_MIN_Jednotky,Report[1].Tolerancia_MAX_Jednotky,Report[1].NameranaHodnota,Report[1].NameranaHodnota_Jednotky,Report[1].VyslednyResult, ADR(TRCB_P2_Maticovacka_ST4.INPUTS.Report));

                Report[2].PoradoveCislo:= '3';
                Report[2].Popis:= 'MaticaM4_CasSrobovania';
                Report[2].FormatHodnoty:= '1';
                Report[2].Tolerancia_MIN_Hodnota:= '';
                Report[2].Tolerancia_MAX_Hodnota:= '';
                Report[2].Nominal:= '';
                Report[2].Tolerancia_MIN_Jednotky:= '';
                Report[2].Tolerancia_MAX_Jednotky:= '';
                Report[2].NameranaHodnota:= Reports.Skrutkovacky.CasSkrutkovania.P2_MaticaM4;
                Report[2].NameranaHodnota_Jednotky:= 's';
                Report[2].VyslednyResult:= Reports.Skrutkovacky.VyslednyReport.P2_MaticaM4;
                SKTcpClientNewCsvEntry(Report[2].PoradoveCislo,Report[2].Popis,Report[2].FormatHodnoty,Report[2].Tolerancia_MIN_Hodnota,Report[2].Tolerancia_MAX_Hodnota,Report[2].Nominal,Report[2].Tolerancia_MIN_Jednotky,Report[2].Tolerancia_MAX_Jednotky,Report[2].NameranaHodnota,Report[2].NameranaHodnota_Jednotky,Report[2].VyslednyResult, ADR(TRCB_P2_Maticovacka_ST4.INPUTS.Report));

                Report[3].PoradoveCislo:= '4';
                Report[3].Popis:= 'MaticaM4_VyskaSrobovania';
                Report[3].FormatHodnoty:= '1';
                Report[3].Tolerancia_MIN_Hodnota:= '';
                Report[3].Tolerancia_MAX_Hodnota:= '';
                Report[3].Nominal:= '';
                Report[3].Tolerancia_MIN_Jednotky:= '';
                Report[3].Tolerancia_MAX_Jednotky:= '';
                Report[3].NameranaHodnota:= Reports.Skrutkovacky.VyskaSkrutkovania.P2_MaticaM4;
                Report[3].NameranaHodnota_Jednotky:= 'mm';
                Report[3].VyslednyResult:= Reports.Skrutkovacky.VyslednyReport.P2_MaticaM4;
                SKTcpClientNewCsvEntry(Report[3].PoradoveCislo,Report[3].Popis,Report[3].FormatHodnoty,Report[3].Tolerancia_MIN_Hodnota,Report[3].Tolerancia_MAX_Hodnota,Report[3].Nominal,Report[3].Tolerancia_MIN_Jednotky,Report[3].Tolerancia_MAX_Jednotky,Report[3].NameranaHodnota,Report[3].NameranaHodnota_Jednotky,Report[3].VyslednyResult, ADR(TRCB_P2_Maticovacka_ST4.INPUTS.Report));

                //Kamera 9//
                Report[4].PoradoveCislo:= '5';
                Report[4].Popis:= 'KAM_9_KontrolaPaletky';
                Report[4].FormatHodnoty:= '2';
                Report[4].Tolerancia_MIN_Hodnota:= '';
                Report[4].Tolerancia_MAX_Hodnota:= '';
                Report[4].Nominal:= 'OK';
                Report[4].Tolerancia_MIN_Jednotky:= '';
                Report[4].Tolerancia_MAX_Jednotky:= '';
                IF Reports.Kamery.P2_CAM9_KontrolaPaletky = 'PASS' THEN
                    Report[4].NameranaHodnota:= 'OK';
                ELSE
                    Report[4].NameranaHodnota:= 'NG';
                END_IF
                Report[4].NameranaHodnota_Jednotky:= '';
                Report[4].VyslednyResult:= Reports.Kamery.P2_CAM9_KontrolaPaletky;
                SKTcpClientNewCsvEntry(Report[4].PoradoveCislo,Report[4].Popis,Report[4].FormatHodnoty,Report[4].Tolerancia_MIN_Hodnota,Report[4].Tolerancia_MAX_Hodnota,Report[4].Nominal,Report[4].Tolerancia_MIN_Jednotky,Report[4].Tolerancia_MAX_Jednotky,Report[4].NameranaHodnota,Report[4].NameranaHodnota_Jednotky,Report[4].VyslednyResult, ADR(TRCB_P2_Maticovacka_ST4.INPUTS.Report));
                SC_KOM_Server.Switch1:= TRUE;
            END_IF

			TRCB_P2_Maticovacka_ST4.INPUTS.CisloPaletky:= 'Pal';
			brsstrcat(ADR(TRCB_P2_Maticovacka_ST4.INPUTS.CisloPaletky), ADR(P2_StoperMaticovacky.PAR.CisloPaletky_STRING));

			TRCB_P2_Maticovacka_ST4.INPUTS.TYP_Prikazu:= '2';
			TRCB_P2_Maticovacka_ST4.INPUTS.CisloStanice:= 'ST4';
			TRCB_P2_Maticovacka_ST4.INPUTS.QRkodPowerCP:= Paletka[a].PAR.QRkodPowerCP;
			TRCB_P2_Maticovacka_ST4.INPUTS.QRkodFiltra:= '';
			TRCB_P2_Maticovacka_ST4.INPUTS.ID_Operatora:= Paletka[a].PAR.ID_Operatora;
			TRCB_P2_Maticovacka_ST4.INPUTS.StavPaletky:= Paletka[a].PAR.StavPowerCP;

			IF SKTcpClientTrace_1.Status.staReadyToSend AND NOT SKTcpClientTrace_1.Cmd.Close THEN
				TRCB_P2_Maticovacka_ST4.OUTPUTS.TYP_Prikazu:= '';
				SKTcpClientTrace_1.Cmd.Send:= TRUE;
				SC_KOM_Server.ResetStep:= TRUE;
				SC_KOM_Server.Step:= 43;
			END_IF

		43:
			SC_KOM_Server.StepName:= '43 - Odoslanie stavu paletky - odpoved servera';
			SC_KOM_Server.IdleTime.PT:= T#3s;
			SC_KOM_Server.AlarmTime.PT:= T#7s;
            SC_KOM_Server.AlarmTime.IN:= TRUE;

			IF SKTcpClientTrace_1.Status.staReceived AND
				(TRCB_P2_Maticovacka_ST4.OUTPUTS.TYP_Prikazu = TRCB_P2_Maticovacka_ST4.INPUTS.TYP_Prikazu) AND
				(TRCB_P2_Maticovacka_ST4.OUTPUTS.QRkodPowerCP = TRCB_P2_Maticovacka_ST4.INPUTS.QRkodPowerCP) THEN
				TRCB_P2_Maticovacka_ST4.STATUS.KomunikaciaUkoncena:= TRUE;
				SC_KOM_Server.ResetStep:= TRUE;
                SC_KOM_Server.Step:= 45;
            ELSIF SC_KOM_Server.AlarmTime.Q AND NOT SKTcpClientTrace_1.Status.staSending THEN
                PocetDopytovNaServer:= PocetDopytovNaServer + 1;
				SKTcpClientTrace_1.Cmd.Close:= TRUE;
				SKTcpClientTrace_1.Cmd.Send:= FALSE;
				SC_KOM_Server.ResetStep:= TRUE;
                SC_KOM_Server.Step:= 44;
			END_IF

        44:
            SC_KOM_Server.StepName:= '44 - Odoslanie stavu paletky - cakam na opatovny dopyt na server';
            SC_KOM_Server.IdleTime.PT:= T#1s;
            SC_KOM_Server.AlarmTime.PT:= T#10s;
            SC_KOM_Server.IdleTime.IN:= TRUE;
            SKTcpClientTrace_1.Cmd.Send:= FALSE;

            IF PocetDopytovNaServer < 3 THEN
                IF SC_KOM_Server.IdleTime.Q THEN
                    SC_KOM_Server.ResetStep:= TRUE;
                    SC_KOM_Server.Step:= 40;
                END_IF
            ELSE
                TRCB_P2_Maticovacka_ST4.STATUS.KomunikaciaError:= TRUE;
                SC_KOM_Server.ResetStep:= TRUE;
                SC_KOM_Server.Step:= 45;
            END_IF

		45:
			SC_KOM_Server.StepName:= '45 - Vyziadanie serioveho cisla - cakam na ukoncenie komunikacie';
			SC_KOM_Server.IdleTime.PT:= T#3s;
			SC_KOM_Server.AlarmTime.PT:= T#10s;

			IF NOT TRCB_P2_Maticovacka_ST4.CMD.OdosliStavPaletky_TYP2 THEN
                SC_KOM_Server.ResetStep:= TRUE;
				SC_KOM_Server.Step:= 0;
			END_IF

		50:
			SC_KOM_Server.StepName:= '50 - Vyziadanie stavu Panatrace - odoslanie dat na server';
			SC_KOM_Server.IdleTime.PT:= T#3s;
			SC_KOM_Server.AlarmTime.PT:= T#10s;
			SC_KOM_Server.AlarmTime.IN:= TRUE;

			TRCB_P2_Maticovacka_ST4.INPUTS.TYP_Prikazu:= '4';
			TRCB_P2_Maticovacka_ST4.INPUTS.CisloStanice:= 'ST4';
			TRCB_P2_Maticovacka_ST4.INPUTS.CisloPaletky:= '';
			TRCB_P2_Maticovacka_ST4.INPUTS.QRkodPowerCP:= '';
			TRCB_P2_Maticovacka_ST4.INPUTS.QRkodFiltra:= '';
			TRCB_P2_Maticovacka_ST4.INPUTS.ID_Operatora:= '';
			TRCB_P2_Maticovacka_ST4.INPUTS.Report:= '';
			TRCB_P2_Maticovacka_ST4.INPUTS.StavPaletky:= '';

			IF SKTcpClientTrace_1.Status.staReadyToSend AND NOT SKTcpClientTrace_1.Cmd.Close THEN
				TRCB_P2_Maticovacka_ST4.OUTPUTS.TYP_Prikazu:= '';
				SKTcpClientTrace_1.Cmd.Send:= TRUE;
				SC_KOM_Server.ResetStep:= TRUE;
				SC_KOM_Server.Step:= 53;
			END_IF

		53:
			SC_KOM_Server.StepName:= '53 - Vyziadanie stavu paletky - odpoved servera';
			SC_KOM_Server.IdleTime.PT:= T#30s;
			SC_KOM_Server.AlarmTime.PT:= T#7s;
			SC_KOM_Server.AlarmTime.IN:= TRUE;

			IF SKTcpClientTrace_1.Status.staReceived AND TRCB_P2_Maticovacka_ST4.OUTPUTS.TYP_Prikazu = TRCB_P2_Maticovacka_ST4.INPUTS.TYP_Prikazu THEN
				TRCB_P2_Maticovacka_ST4.STATUS.KomunikaciaUkoncena:= TRUE;
				SC_KOM_Server.ResetStep:= TRUE;
				SC_KOM_Server.Step:= 55;
			ELSIF SC_KOM_Server.AlarmTime.Q AND NOT SKTcpClientTrace_1.Status.staSending THEN
				PocetDopytovNaServer:= PocetDopytovNaServer + 1;
				SKTcpClientTrace_1.Cmd.Close:= TRUE;
				SKTcpClientTrace_1.Cmd.Send:= FALSE;
				SC_KOM_Server.ResetStep:= TRUE;
				SC_KOM_Server.Step:= 54;
			END_IF

		54:
			SC_KOM_Server.StepName:= '54 - Vyziadanie stavu paletky - cakam na opatovny dopyt na server';
			SC_KOM_Server.IdleTime.PT:= T#1s;
			SC_KOM_Server.AlarmTime.PT:= T#10s;
			SC_KOM_Server.IdleTime.IN:= TRUE;

			IF PocetDopytovNaServer < 3 THEN
				IF SC_KOM_Server.IdleTime.Q THEN
					SC_KOM_Server.ResetStep:= TRUE;
					SC_KOM_Server.Step:= 50;
				END_IF
			ELSE
				TRCB_P2_Maticovacka_ST4.STATUS.KomunikaciaError:= TRUE;
				SC_KOM_Server.ResetStep:= TRUE;
				SC_KOM_Server.Step:= 55;
			END_IF

		55:
			SC_KOM_Server.StepName:= '55 - Vyziadanie stavu paletky - cakam na ukoncenie komunikacie';
			SC_KOM_Server.IdleTime.PT:= T#3s;
			SC_KOM_Server.AlarmTime.PT:= T#10s;

			IF NOT TRCB_P2_Maticovacka_ST4.CMD.VyziadajStavPanatrace_TYP4 THEN
				SC_KOM_Server.ResetStep:= TRUE;
				SC_KOM_Server.Step:= 0;
			END_IF

	END_CASE

END_PROGRAM

PROGRAM _EXIT
	(* Insert code here *)

END_PROGRAM
```

#### Types.typ - Local data types
```iecst
TYPE
	Report_typ : 	STRUCT
		PoradoveCislo : STRING[2]; (*IDstep - Poradové čislo reportu*)
		Popis : STRING[100]; (*Description - Popis*)
		FormatHodnoty : STRING[2]; (*TypValue - Format zaslané hodnoty  1- Číslo, 2 - Znak*)
		Tolerancia_MIN_Hodnota : STRING[10]; (*MinTol - Minimálna tolerancia meranej veličiny*)
		Tolerancia_MAX_Hodnota : STRING[10]; (*MaxTol - Maximálna tolerancia meranej veličiny*)
		Nominal : STRING[10]; (*Nom - Ak jezvolený formát string tak tu zadáme OK inak je prazdna*)
		Tolerancia_MIN_Jednotky : STRING[10]; (*MinEle - Jednotky minimálnej tolerancie veličiny*)
		Tolerancia_MAX_Jednotky : STRING[10]; (*MaxEle - Jednotky maximálnej tolerancie veličiny*)
		NameranaHodnota : STRING[10]; (*Value - Namerana hodnota veličiny, ak su kamery tak bude hodnota OK alebo NG*)
		NameranaHodnota_Jednotky : STRING[10]; (*ValEle - Jednotky nameranej veličiny*)
		VyslednyResult : STRING[5]; (*Result - Výsledný result  PASS, FAIL, SKIP*)
	END_STRUCT;
END_TYPE
```

#### Variables.var - Local variables
```iecst
VAR
	SC_KOM_Server : SequenceControlTyp;
	SKTcpClientTrace_1 : SKTcpClientTrace;
	a : USINT;
	Report : ARRAY[0..50] OF Report_typ;
	PocetDopytovNaServer : USINT;
END_VAR
```

### Program Logical/TracebilitySystem/P2_Srobovanie_ST5 (IEC)
